PROGRAM UN01
VAR
	Ref_Unit: REFERENCE TO UDT_UnitAdmin;
	Ref_MachineStateModel: REFERENCE TO PackMlv3_StateModel;
	ref_Master1: REFERENCE TO UDT_AXISADMIN;	
	Cfg_ModeNames: ARRAY[0..31] OF STRING;
	Cfg_DisableStates: ARRAY [0..31] OF DINT;
	Cfg_ModeTransitions: ARRAY [0..31] OF DINT;
	HMI_O_StateCurrentName: STRING(255);
	HMI_O_ModeCurrentName: STRING(255);
	iHmiErr: INT;
	Loc_diEM_AbortingDone: DINT;
	Loc_diEM_ClearingDone: DINT;
	Loc_diEM_HoldingDone: DINT;
	Loc_diEM_ResettingDone: DINT;
	Loc_diEM_StartingDone: DINT;
	Loc_diEM_StoppingDone: DINT;
	Loc_diEM_SuspendingDone: DINT;
	Loc_diEM_UnSuspendingDone: DINT;
	Loc_diEM_UnHoldingDone: DINT;	
	Loc_diEM_Fault: DINT;
	Loc_diEM_Warning: DINT;	

	// 安全复位
	tonSafetyReset: TON;
	ft_SafetyReset: F_TRIG;
	iSafetyResetSeq: INT;	
	//EtherCat	
	iFaultClearSeq: INT;
	tonFaultClear: Ton;
	bClearAllFault: BOOL;
	xDebugReset: BOOL;
	arEventEmpty: ARRAY[1..256] OF BOOL;
	arSys1EventEmpty: ARRAY[1..20] OF BOOL;
	arSys2EventEmpty: ARRAY[21..40] OF BOOL;
	arSys3EventEmpty: ARRAY[1..20] OF BOOL;	
	loc_bAnyStopError: BOOL;
	j: INT;

	tonTimeHigh: TON;
	tonTimeLow: TON;
	arBlink: ARRAY[1..10] OF blink;
	
	tonFaultHandler: Ton;	
	StopEvent: ARRAY[0..40] OF UDT_EVENT;	
	arCylinder_AOI: ARRAY[1..80] OF AOI_CylinderAdmin;	
	arVacuum_AOI: ARRAY[1..60] OF AOI_VacuumAdmin;
    arSensor_AOI: ARRAY[1..60] OF AOI_Sensoradmin;	
	arHeat_AOI: ARRAY[1..8] OF Aoi_HeatBase;
    bUnitFS: BOOL;

	diUnitStopEvent0: DINT;
	rtWorkLocMode: R_trig;
	iRecipeSeq: INT;
	tonCmdReset: TON;
	tonCmdStart: TON;
	diSys1StopEvent1: DINT;
	diSys1StopEvent2: DINT;
	diSys2StopEvent1: DINT;
	diSys2StopEvent2: DINT;
	diSys3StopEvent1: DINT;
	diSys3StopEvent2: DINT;
	diSys3StopEvent3: DINT;
	rtAllaxisHomed: R_TRIG;
	tonRecipeSeq: Ton;
	
	tongeneralEvent0:ARRAY[0..255] OF Ton;

	diSys3StopEvent4: DINT;
	bSys1StopError: BOOL;
	bSys2StopError: BOOL;
	bSys3StopError: BOOL;

	iC: INT;
	
	arDropCylinder_AOI: ARRAY[1..40] OF AOI_CylinderAdmin;	
	iNotDone: INT;
	aoiActiveTotalTime: AOI_Timer;
	aoiWorkTotalTime: AOI_Timer;
	aoi10MinuteTime: AOI_Timer;
	
	rtGoodCount: R_TRIG;
	rtNoGoodCount: R_trig;
	rMaxCounterTime: DINT;
	rMaxDropTime: DINT;
	i: INT;
	iInitCnt: INT;
	iAutoCut: INT;
	tonAutoCut: Ton;
	iCutCnt: INT;
	bBoxRecipeUpdate: BOOL;
	bEn10Minute: BOOL;
	bReset10Minute: BOOL;
	diTransferCntOld: DINT;
	tonRecipeReset: Ton;
	bFirstCyclinderScan: BOOL;
	bAnySaftyDoorOpen: BOOL;
	tonCounterAirOpen: Ton;
END_VAR

VAR CONSTANT
   EM_OK: ARRAY[0..64] OF BOOL :=[65(0)];
   diEm_Done: DINT:=0;
END_VAR

//PLC IP地址IP 192.168.1.10 HMI1 IP 192.168.1.12 HMI2 IP 192.168.1.13 路由器 192.168.1.1 密码IPB19021 账号admin
//plc administrator 1 
//HMI 2222 
//激光打标机IP 192.168.1.20 
Ref_Unit REF=Unit01;
Ref_MachineStateModel REF= UN01_MachineStateModel;
ref_Master1 REF= arVirtualAxisAdmin[1];
CM02_ConditionsModules();
CM03_Cylinder();
CM04_Vacuum();
CM05_Sensor();
CM06_Heat();
CM07_Counters();
CM10_LightStatus();
SR02_Recipe();
UP01_PackML();
UP02_StateComplete();
EM01_Master();
EM02_Follower1();
EM03_Follower2();
EM04_FOllower3();
EM05_Counters();
EM06_Follower4_5();
EM07_Belt6();
EM08_Belt7();
SR91_OEE();
CM01_OperationLocal();
SR05_Manual();

IF NOT bUnitFS THEN
   SR01_Initialize();
END_IF

SR03_FaultHandler();
SR04_Parameter();
SR90_SafetyReset();
SR99_FaultClear();

DebugPro();

ACTION CM01_OperationLocal:
Ref_MachineStateModel.Cmd_Clear:=HMI_LocModeInput.ClearFault OR xDebugReset;
bAnySaftyDoorOpen:=arSafeDoorSts[19] OR arSafeDoorSts[20] OR arSafeDoorSts[21] OR arSafeDoorSts[22];
//前后设备急停串联
IF (glb_diEstopButton_UN01<>0) THEN
	Ref_MachineStateModel.Cmd_Abort:=TRUE;
	glb_AllAxisHomed_UN01:=FALSE;
	ELSE
	Ref_MachineStateModel.Cmd_Abort:=FALSE;
END_IF
//清除故障
IF Ref_MachineStateModel.Cmd_Clear THEN
   bClearAllFault:=TRUE;
END_IF
//停机
IF (HMI_LocModeInput.Stop OR glb_bStopButton_UN01) OR 
   (bAnySaftyDoorOpen AND Ref_MachineStateModel.Sts_Resetting) AND NOT Ref_MachineStateModel.Sts_Held THEN
	Ref_MachineStateModel.Cmd_Stop:=TRUE;
	ELSE
	Ref_MachineStateModel.Cmd_Stop:=FALSE;	
END_IF
//暂停
IF ((loc_bAnyStopError OR bAnySaftyDoorOpen) AND Ref_MachineStateModel.Sts_Execute) 
OR HMI_LocModeInput.Hold THEN
	Ref_MachineStateModel.Cmd_Hold:=TRUE;
	ELSE
	Ref_MachineStateModel.Cmd_Hold:=FALSE;	
END_IF
//启动
tonCmdStart(IN:= (HMI_LocModeInput.Start OR glb_bStartButton_UN01), PT:=T#2S , Q=> , ET=> );
IF tonCmdStart.Q AND glb_bAllSafetyOk 
AND NOT loc_bAnyStopError  
AND Ref_MachineStateModel.Sts_Idle
AND glb_bModeSwitch_UN01 THEN
	Ref_MachineStateModel.Cmd_Start:=TRUE;
	ELSE
	Ref_MachineStateModel.Cmd_Start:=FALSE;	
END_IF
//复位
tonCmdReset(IN:= (HMI_LocModeInput.Reset OR glb_bResetButton_UN01), PT:=T#2S , Q=> , ET=> );
IF tonCmdReset.Q AND NOT loc_bAnyStopError AND glb_bModeSwitch_UN01 THEN
   IF HMI_LocModeINPUT.Reset THEN
	  glb_AllAxisHomed_UN01:=FALSE;
   END_IF
   Ref_MachineStateModel.Cmd_Reset:=TRUE;
   ELSE
   Ref_MachineStateModel.Cmd_Reset:=FALSE;	 
END_IF

//安全复位
IF (glb_bResetButton_UN01 OR glb_bResetButton_UN02) AND
NOT glb_bAllSafetyOk THEN
   glb_bSafetyReset:=TRUE;
END_IF

//解除暂停
IF tonCmdStart.Q  AND Ref_MachineStateModel.Sts_Held  
AND glb_bModeSwitch_UN01 AND NOT loc_bAnyStopError THEN
	Ref_MachineStateModel.Cmd_UnHold:=TRUE;
	ELSE
    Ref_MachineStateModel.Cmd_UnHold:=FALSE;
END_IF

//等待启动
IF Ref_MachineStateModel.Sts_Idle THEN
	glb_AllAxisHomed_UN01:=TRUE;
END_IF
END_ACTION

ACTION CM02_ConditionsModules:
Loc_diEM_AbortingDone:=MEMCMP(pBuf1:=ADR(Ref_Unit.EM_Aborting_Done) , pBuf2:=ADR(Ref_Unit.EM_Selected) , n:=SIZEOF(Ref_Unit.EM_Selected));
Loc_diEM_ClearingDone:=MEMCMP(pBuf1:=ADR(Ref_Unit.EM_Clearing_Done) , pBuf2:=ADR(Ref_Unit.EM_Selected) , n:=SIZEOF(Ref_Unit.EM_Selected));
Loc_diEM_HoldingDone:=MEMCMP(pBuf1:=ADR(Ref_Unit.EM_Holding_Done) , pBuf2:=ADR(Ref_Unit.EM_Selected) , n:=SIZEOF(Ref_Unit.EM_Selected));
Loc_diEM_ResettingDone:=MEMCMP(pBuf1:=ADR(Ref_Unit.EM_Resetting_Done) , pBuf2:=ADR(Ref_Unit.EM_Selected) , n:=SIZEOF(Ref_Unit.EM_Selected));
Loc_diEM_StartingDone:=MEMCMP(pBuf1:=ADR(Ref_Unit.EM_Starting_Done) , pBuf2:=ADR(Ref_Unit.EM_Selected) , n:=SIZEOF(Ref_Unit.EM_Selected));
Loc_diEM_StoppingDone:=MEMCMP(pBuf1:=ADR(Ref_Unit.EM_Stopping_Done) , pBuf2:=ADR(Ref_Unit.EM_Selected) , n:=SIZEOF(Ref_Unit.EM_Selected));
Loc_diEM_SuspendingDone:=MEMCMP(pBuf1:=ADR(Ref_Unit.EM_Suspending_Done) , pBuf2:=ADR(Ref_Unit.EM_Selected) , n:=SIZEOF(Ref_Unit.EM_Selected));
Loc_diEM_UnSuspendingDone:=MEMCMP(pBuf1:=ADR(Ref_Unit.EM_UnSuspending_Done) , pBuf2:=ADR(Ref_Unit.EM_Selected) , n:=SIZEOF(Ref_Unit.EM_Selected));
Loc_diEM_UnHoldingDone:=MEMCMP(pBuf1:=ADR(Ref_Unit.EM_UnHolding_Done) , pBuf2:=ADR(Ref_Unit.EM_Selected) , n:=SIZEOF(Ref_Unit.EM_Selected));

Loc_diEM_Fault:=MEMCMP(pBuf1:=ADR(Ref_Unit.EM_Fault) , pBuf2:=ADR(EM_OK) , n:=SIZEOF(Ref_Unit.EM_Selected));
Loc_diEM_Warning:=MEMCMP(pBuf1:=ADR(Ref_Unit.EM_Warning) , pBuf2:=ADR(EM_OK) , n:=SIZEOF(Ref_Unit.EM_Selected));

Ref_Unit.EM_Selected:=HMI_EMSelectUn01;
END_ACTION

ACTION CM03_Cylinder:
FOR i:= 1 TO 60 DO
	arPackCylinder[i].i.CheckTime:=10000;
	arPackCylinder[i].i.Mode:=1;	
    arCylinder_AOI[i](Admin:= arPackCylinder[i]);
END_FOR
	arDropBufferCyclinder[1].i.CheckTime:=10000;
	arDropBufferCyclinder[1].i.Mode:=1;
	arDropBufferCyclinder[2].i.CheckTime:=10000;
	arDropBufferCyclinder[2].i.Mode:=1;
arCylinder_AOI[61](Admin:= arDropBufferCyclinder[1]);
arCylinder_AOI[62](Admin:= arDropBufferCyclinder[2]);
IF NOT bFirstCyclinderScan THEN
   bFirstCyclinderScan:=TRUE;
END_IF
END_ACTION

ACTION CM04_Vacuum:
FOR i:=1 TO 60 DO
	arPackVacuum[i].i.CheckTime:=5000;
	arPackVacuum[i].i.BlowTime:=1000;
	arVacuum_AOI[i](admin:= arPackVacuum[i]);
END_FOR
END_ACTION

ACTION CM05_Sensor:
FOR i:=1 TO 60 DO
	arSensor_AOI[i](Admin:=arPackSensor[i] );
END_for
END_ACTION

ACTION CM06_Heat:
	arHeat_AOI[1](	Enable:=NOT HMI_HeatDisable , 	PV:=HMI_HeatTempAct[1] , 	SV:= HMI_HeatTempSet[1], 
 	Reset:= ,HighLimit:= 30,lowLimit:= 30,MaxLimit:=300,Kp:=20,Ki:=0.5,Kd:=3,
	Active=> arPackHeatRealy[1], 
	Error=> );
	arHeat_AOI[2](	Enable:=NOT HMI_HeatDisable , 	PV:=HMI_HeatTempAct[2] , 	SV:= HMI_HeatTempSet[2], 
	Reset:= ,HighLimit:= 30, lowLimit:= 30,MaxLimit:=300,Kp:=20,Ki:=0.5,Kd:=3,
	Active=> arPackHeatRealy[2], 
	Error=> );
	arHeat_AOI[3](	Enable:=NOT HMI_HeatDisable , 	PV:=HMI_HeatTempAct[3] , 	SV:= HMI_HeatTempSet[3], 
    Reset:= ,HighLimit:= 30, lowLimit:= 30,MaxLimit:=300,Kp:=20,Ki:=0.5,Kd:=3,
	Active=> arPackHeatRealy[3], 
	Error=> );
	arHeat_AOI[4](	Enable:=NOT HMI_HeatDisable , 	PV:=HMI_HeatTempAct[4] , 	SV:= HMI_HeatTempSet[4], 
    Reset:= ,HighLimit:= 30, lowLimit:= 30,MaxLimit:=300,Kp:=20,Ki:=0.5,Kd:=3,		
	Active=> arPackHeatRealy[4], 
	Error=> );
	arHeat_AOI[5](	Enable:=NOT HMI_HeatDisable , 	PV:=HMI_HeatTempAct[5] , 	SV:= HMI_HeatTempSet[5], 
    Reset:= ,HighLimit:= 30, lowLimit:= 30,MaxLimit:=300,Kp:=20,Ki:=0.5,Kd:=3,		
	Active=> arPackHeatRealy[5], 
	Error=> );
	arHeat_AOI[6](	Enable:=NOT HMI_HeatDisable , 	PV:=HMI_HeatTempAct[6] , 	SV:= HMI_HeatTempSet[6],
    Reset:= ,HighLimit:= 30, lowLimit:= 30,MaxLimit:=300,Kp:=20,Ki:=0.5,Kd:=3, 
	Active=> arPackHeatRealy[6], 
	Error=> );
	arHeat_AOI[7](	Enable:=NOT HMI_HeatDisable , 	PV:=HMI_HeatTempAct[7] , 	SV:= HMI_HeatTempSet[7],
    Reset:= ,HighLimit:= 30, lowLimit:= 30,MaxLimit:=300,Kp:=20,Ki:=0.5,Kd:=3, 
	Active=> arPackHeatRealy[7], 
	Error=> );
	arHeat_AOI[8](	Enable:=NOT HMI_HeatDisable , 	PV:=HMI_HeatTempAct[8] , 	SV:= HMI_HeatTempSet[8],
    Reset:= ,HighLimit:= 30, lowLimit:= 30,MaxLimit:=300,Kp:=20,Ki:=0.5,Kd:=3, 
	Active=> arPackHeatRealy[8], 
	Error=> );	
	
	HMI_HeatTempAct[1]:=INT_TO_REAL(EL3312[1,1].Value)/10;
	HMI_HeatTempAct[2]:=INT_TO_REAL(EL3312[1,2].Value)/10;
	HMI_HeatTempAct[3]:=INT_TO_REAL(EL3312[2,1].Value)/10;
	HMI_HeatTempAct[4]:=INT_TO_REAL(EL3312[2,2].Value)/10;
	HMI_HeatTempAct[5]:=INT_TO_REAL(EL3312[3,1].Value)/10;
	HMI_HeatTempAct[6]:=INT_TO_REAL(EL3312[3,2].Value)/10;   
	HMI_HeatTempAct[7]:=INT_TO_REAL(EL3312[4,1].Value)/10;
	HMI_HeatTempAct[8]:=INT_TO_REAL(EL3312[4,2].Value)/10;
END_ACTION

ACTION CM07_Counters:
iInitCnt:=0;
rMaxDropTime:=0;
rMaxCounterTime:=0;
FOR ic:=1 TO 10 DO
	arCounters[iC](
		In_Total:= RecipeBuffer.amount, 
		Quantity:= RecipeBuffer.Counters[iC].Quantity, 
		ProcessTime=> HMI_OEEView.CounterProcessTime[iC] ,
		Axis:= arRealAxisAdmin[iC], 
		Checktime:= HMI_CntCheckTime,
		DropSensor:= arDropSensor[iC], 
		LowSensor:= arLowSensor[iC], 
		HighSensor:= arhighSensor[iC],
		DropFlag:= glb_BinBelt1.bin[iC].arDrop[iC],
		Cylinder:= arDropCylinder[iC]);	
END_FOR
FOR ic:=11 TO 20 DO
	arCounters[iC](
		In_Total:= RecipeBuffer.amount, 
		Quantity:= RecipeBuffer.Counters[iC].Quantity,
       	CheckTime:= 1500,
		ProcessTime=> HMI_OEEView.CounterProcessTime[iC] ,
		Axis:= arRealAxisAdmin[iC], 
		Checktime:= HMI_CntCheckTime,
		DropSensor:= arDropSensor[iC], 
		LowSensor:= arLowSensor[iC], 
		HighSensor:= arhighSensor[iC],
		DropFlag:= glb_BinBelt1.bin[iC+20].arDrop[iC+20],
		Cylinder:= arDropCylinder[iC]);	
END_FOR

FOR ic:=21 TO 30 DO
	arCounters[iC](
		In_Total:= RecipeBuffer.amount, 
		Quantity:= RecipeBuffer.Counters[iC].Quantity, 
		ProcessTime=> HMI_OEEView.CounterProcessTime[iC] ,
		Axis:= arRealAxisAdmin[iC], 
		Checktime:= HMI_CntCheckTime,
		DropSensor:= arDropSensor[iC], 
		LowSensor:= arLowSensor[iC], 
		HighSensor:= arhighSensor[iC],
		DropFlag:= glb_BinBelt2.bin[ic-20].arDrop[iC-20],
		Cylinder:= arDropCylinder[iC]);	
END_FOR

FOR ic:=31 TO 40 DO
	arCounters[iC](
		In_Total:= RecipeBuffer.amount, 
		Quantity:= RecipeBuffer.Counters[iC].Quantity, 
		ProcessTime=> HMI_OEEView.CounterProcessTime[iC] ,
		Axis:= arRealAxisAdmin[iC], 
		Checktime:= HMI_CntCheckTime,
		DropSensor:= arDropSensor[iC], 
		LowSensor:= arLowSensor[iC], 
		HighSensor:= arhighSensor[iC],
		DropFlag:= glb_BinBelt2.bin[iC].arDrop[iC],
		Cylinder:= arDropCylinder[iC]);	
END_FOR
  
FOR iC:=1 TO 40 DO
	arDropCylinder_AOI[iC](Admin:= arDropCylinder[iC]);
	arDropCylinder[iC].i.CheckTime:=1500;
	arDropCylinder[iC].i.Mode:=1;	
   IF NOT  arCounters[iC].Busy THEN
      IF rMaxCounterTime < arCounters[iC].ProcessTime THEN
		 rMaxCounterTime:= arCounters[iC].ProcessTime;
	  END_IF
   END_IF  
   arCounters[iC].SkipAlarm:=HMI_SkipCntAlarm[iC];
   arCounters[iC].CheckCnt:=HMI_CntCheck[iC];
   HMI_CountersCntUp[ic]:=arCounters[iC].CntUp;
   
   HMI_OEEView.DropProcessTime[ic]:=(arDropCylinder_AOI[iC].ActInTime+arDropCylinder_AOI[iC].ActOutTime)/2;
   IF rMaxDropTime<HMI_OEEView.DropProcessTime[ic] THEN
	  rMaxDropTime:=HMI_OEEView.DropProcessTime[ic];  
   END_IF
END_FOR
END_ACTION

ACTION CM10_LightStatus:

IF glb_bAllSafetyOk THEN
	glb_bResetBottonLight_UN01:=TRUE;
	ELSE 
    glb_bResetBottonLight_UN01:=arBlink[1].OUT;
END_IF

{region Lihgtsys1} 
//红灯
glb_arLightRed_UN01[1]:=Ref_MachineStateModel.Sts_Aborted OR Ref_MachineStateModel.Sts_Aborting OR (arblink[1].OUT AND bSys1StopError);
glb_arLightAlarm_UN01[1]:=(glb_arLightRed_UN01[1] OR glb_arLightYellow_UN01[1]) AND NOT HMI_AlarmMute;
//绿灯	  
glb_arLightGreen_UN01[1]:= Ref_MachineStateModel.Sts_Execute OR  Ref_MachineStateModel.Sts_Stopping OR
( arblink[1].OUT AND NOT bSys1StopError  AND NOT Ref_MachineStateModel.Sts_Aborted AND NOT Ref_MachineStateModel.Sts_Resetting
AND( Ref_MachineStateModel.Sts_Stopped OR Ref_MachineStateModel.Sts_Idle OR Ref_MachineStateModel.Sts_Held))
OR (Ref_MachineStateModel.Sts_Resetting  AND arblink[2].OUT);	 
//黄灯
glb_arLightYellow_UN01[1]:= (HMI_GeneralEvent[2].ID[1] OR HMI_GeneralEvent[2].ID[2] OR HMI_GeneralEvent[2].ID[3] OR HMI_GeneralEvent[2].ID[4]
OR HMI_GeneralEvent[2].ID[5] OR HMI_GeneralEvent[2].ID[6] OR HMI_GeneralEvent[2].ID[7] OR HMI_GeneralEvent[2].ID[8] OR HMI_GeneralEvent[2].ID[9]
OR HMI_GeneralEvent[2].ID[10] OR HMI_GeneralEvent[2].ID[11] OR HMI_GeneralEvent[2].ID[12] OR HMI_GeneralEvent[2].ID[13] OR HMI_GeneralEvent[2].ID[14]
OR HMI_GeneralEvent[2].ID[15] OR HMI_GeneralEvent[2].ID[16] OR HMI_GeneralEvent[2].ID[17] OR HMI_GeneralEvent[2].ID[18] OR HMI_GeneralEvent[2].ID[19]
OR HMI_GeneralEvent[2].ID[20]) AND arblink[1].OUT;	 	 
		  
(*照明灯*)  
glb_arLightRelay_UN01[1]:= arSafeDoorSts[1] OR arSafeDoorSts[2] OR arSafeDoorSts[3] OR arSafeDoorSts[4] OR
arSafeDoorSts[5] OR arSafeDoorSts[6] OR arSafeDoorSts[7] OR arSafeDoorSts[8] OR
arSafeDoorSts[9] ;
	   
{end_region}				
{region Lihgtsys2} 					 

glb_arLightRed_UN01[2]:=Ref_MachineStateModel.Sts_Aborted OR Ref_MachineStateModel.Sts_Aborted OR ( arblink[1].OUT AND bSys2StopError );
glb_arLightAlarm_UN01[2]:=(glb_arLightRed_UN01[2] OR glb_arLightYellow_UN01[2]) AND NOT HMI_AlarmMute;
		  
glb_arLightGreen_UN01[2]:= Ref_MachineStateModel.Sts_Execute OR Ref_MachineStateModel.Sts_Stopping OR
( arblink[1].OUT AND NOT bSys2StopError  AND NOT Ref_MachineStateModel.Sts_Aborted AND NOT Ref_MachineStateModel.Sts_Resetting
AND( Ref_MachineStateModel.Sts_Stopped OR Ref_MachineStateModel.Sts_Idle OR Ref_MachineStateModel.Sts_Held))
OR (Ref_MachineStateModel.Sts_Resetting  AND arblink[2].OUT);
 
//黄灯
glb_arLightYellow_UN01[2]:= (HMI_GeneralEvent[2].ID[21] OR HMI_GeneralEvent[2].ID[22] OR HMI_GeneralEvent[2].ID[23] OR HMI_GeneralEvent[2].ID[24]
OR HMI_GeneralEvent[2].ID[25] OR HMI_GeneralEvent[2].ID[26] OR HMI_GeneralEvent[2].ID[27] OR HMI_GeneralEvent[2].ID[28] OR HMI_GeneralEvent[2].ID[29]
OR HMI_GeneralEvent[2].ID[30] OR HMI_GeneralEvent[2].ID[31] OR HMI_GeneralEvent[2].ID[32] OR HMI_GeneralEvent[2].ID[33] OR HMI_GeneralEvent[2].ID[34]
OR HMI_GeneralEvent[2].ID[35] OR HMI_GeneralEvent[2].ID[36] OR HMI_GeneralEvent[2].ID[37] OR HMI_GeneralEvent[2].ID[38] OR HMI_GeneralEvent[2].ID[39]
OR HMI_GeneralEvent[2].ID[40]) AND arblink[1].OUT;		   
(*照明灯*)

glb_arLightRelay_UN01[2]:=arSafeDoorSts[10] OR arSafeDoorSts[11] OR arSafeDoorSts[12] OR arSafeDoorSts[13] OR
arSafeDoorSts[14] OR arSafeDoorSts[15] OR arSafeDoorSts[16] OR arSafeDoorSts[17] OR
arSafeDoorSts[18] ;
	  
{end_region}		   

{region Lihgtsys3} 	

glb_arLightRed_UN01[3]:=Ref_MachineStateModel.Sts_Aborted OR Ref_MachineStateModel.Sts_Aborted OR (arblink[1].OUT AND bSys3StopError);
glb_arLightAlarm_UN01[3]:=glb_arLightRed_UN01[3] AND NOT HMI_AlarmMute;
			   
							  
glb_arLightGreen_UN01[3]:= Ref_MachineStateModel.Sts_Execute OR Ref_MachineStateModel.Sts_Stopping OR
( arblink[1].OUT AND NOT bSys3StopError  AND NOT Ref_MachineStateModel.Sts_Aborted AND NOT Ref_MachineStateModel.Sts_Resetting
AND( Ref_MachineStateModel.Sts_Stopped OR Ref_MachineStateModel.Sts_Idle OR Ref_MachineStateModel.Sts_Held))
OR (Ref_MachineStateModel.Sts_Resetting  AND arblink[2].OUT);
//黄灯
glb_arLightYellow_UN01[3]:= ( HMI_GeneralEvent[0].ID[1] OR HMI_GeneralEvent[0].ID[2] ) AND arblink[1].OUT;		   
(*照明灯*)

{end_region}

arBlink[1](TimeH:=100 , TimeL:=1000 , OUT=> );
arBlink[2](TimeH:=200 , TimeL:=200 , OUT=> );
END_ACTION

ACTION SR01_Initialize:
glb_bCounterAirValve_UN01:=TRUE;
bUnitFS:=TRUE;
HMI_EMSelectUN01[1]:=TRUE;
HMI_EMSelectUN01[2]:=TRUE;
HMI_EMSelectUN01[3]:=TRUE;
HMI_EMSelectUN01[4]:=TRUE;
HMI_EMSelectUN01[5]:=TRUE;
HMI_EMSelectUN01[6]:=TRUE;
HMI_EMSelectUN01[7]:=TRUE;
HMI_EMSelectUN01[8]:=TRUE;
	
;
END_ACTION

ACTION SR02_Recipe:
rtWorkLocMode(CLK:=HMI_LocModeEnable , Q=> );
rtAllaxisHomed(CLK:= glb_AllAxisHomed_UN01, Q=> );
tonRecipeReset(IN:=glb_bResetButton_UN01 AND Ref_MachineStateModel.Sts_Execute , PT:= T#5S , Q=> , ET=> );

CASE iRecipeSeq OF 
	0: 
	   HMI_RecipeReset:=TRUE;
	   bBoxRecipeUpdate:=FALSE;
       IF  glb_AllAxisHomed_UN01  THEN
		   IF HMI_LocModeEnable THEN
			  iRecipeSeq:=10;
		   END_IF
		   IF Hmi_Input.ModifyRecipe OR tonRecipeReset.Q THEN 
			  iRecipeSeq:=20;
			  HMI_RecipeReset:=FALSE;
		   END_IF
		   IF HMI_RecipeRedo THEN
			  HMI_RecipeReset:=FALSE;
			  iRecipeSeq:=300;  
		   END_IF
		   IF HMI_RecipCancel THEN
			  HMI_RecipeReset:=FALSE;
			  iRecipeSeq:=200;  
		   END_IF
	   END_IF
	
	10:(*本地模拟生产配方*)
        Hmi_Output.InQuantity:=49;
		Hmi_Output.OutQuantity:=0;
		FOR i:=1 TO 40 DO
			Hmi_Output.Counters[i].Quantity:=5;
			Hmi_Output.Counters[i].ID:=i;
		END_FOR
	    iRecipeSeq:=90;	


     20:
        (**生产任务配方**)
		IF Hmi_Recipe.amount<>0 THEN//配方有效
			RecipeBuffer:=HMI_RECIPE;
			RecipeBuffer.user:=HMI_RECIPE.user;
			Hmi_Output.InQuantity:=RecipeBuffer.amount;
			Hmi_Output.OutQuantity:=0;
			FOR i:=1 TO 40 DO
				Hmi_Output.Counters[i].Quantity:=RecipeBuffer.Counters[i].Quantity;
				Hmi_Output.Counters[i].ID:=RecipeBuffer.Counters[i].ID;
			END_FOR
			iRecipeSeq:=90;	
		ELSE//配方无效
            iRecipeSeq:=200;	
		END_IF
 

		
	90: //复位料仓
        Glb_BinList.Reset:=TRUE;
		FOR i:=1 TO 40 DO
		    arCounters[i].Reset:=TRUE;
		END_FOR 
	    iRecipeSeq:=91;
    91: //复位数粒 		
		FOR i:=1 TO 40 DO
		    arCounters[i].Reset:=FALSE;
		END_FOR
		Glb_BinList.Reset:=FALSE;
		glb_lrMasterTargetCnt:=glb_lrMasterTargetCnt + Hmi_Output.InQuantity;
		glb_lrBelt1TargetCnt:=glb_lrBelt1TargetCnt + Hmi_Output.InQuantity + HMI_B1DropBinNo;
		glb_lrBelt2Targetcnt:=glb_lrBelt2Targetcnt + Hmi_Output.InQuantity + HMI_B2DropBinNo;
		glb_lrBelt3Targetcnt:=glb_lrBelt3Targetcnt+ Hmi_Output.InQuantity + HMI_B3DropBinNo3;	
		iRecipeSeq:=92;
		
	92:	
	    tonRecipeSeq(IN:=TRUE, PT:=T#1S , Q=> , ET=> );
		IF tonRecipeSeq.Q THEN
	       tonRecipeSeq(IN:=FALSE, PT:=T#1S , Q=> , ET=> );	
			HMI_Output.RecipeComplete:=FALSE;
			Hmi_Input.ModifyRecipe:=FALSE;
			HMI_Output.RecipeModifyDone:=TRUE;	  	  
            iRecipeSeq:=93;	
		END_IF	
		
	93:
        tonRecipeSeq(IN:=TRUE, PT:=T#1S , Q=> , ET=> );
		IF tonRecipeSeq.Q THEN
	       tonRecipeSeq(IN:=FALSE, PT:=T#1S , Q=> , ET=> );	  	  
           iRecipeSeq:=100;	
		END_IF	
	 
	100:
	    glb_BinBelt1.bin[1].Name:=RecipeBuffer.user;
		glb_BinBelt1.bin[1].Amount:=RecipeBuffer.amount;//获取生产数量
	    HMI_RecipeAbort:=FALSE;
        Hmi_Output.RecipeEmplty:=FALSE;
		IF glb_lrBelt1wrkCnt>14  AND NOT bBoxRecipeUpdate  THEN
		   glb_lrBoxTargetCnt := glb_lrBoxTargetCnt+Hmi_Output.InQuantity/7;
		   bBoxRecipeUpdate:=TRUE;
		END_IF

		IF glb_lrBelt1wrkCnt = glb_lrBelt1TargetCnt AND glb_lrBelt2wrkCnt = glb_lrBelt2TargetCnt THEN
			HMI_Output.RecipeComplete:=TRUE;
		END_IF
		
	    IF HMI_Output.RecipeComplete THEN
		   HMI_Output.RecipeModifyDone:=FALSE;
	       iRecipeSeq:=110;
		   ELSE IF NOT glb_AllAxisHomed_UN01 THEN//配方被中止
			           HMI_RecipeAbort:=TRUE;
					   iRecipeSeq:=900;
		        END_IF
		END_IF
		
    
    110:
	    tonRecipeSeq(IN:=TRUE, PT:=T#1S , Q=> , ET=> );
		IF tonRecipeSeq.Q THEN
	       tonRecipeSeq(IN:=FALSE, PT:=T#1S , Q=> , ET=> );	
           iRecipeSeq:=0;		
		END_IF
		
(***************************************************************)		
    200: 
        HMI_RecipeAbort:=FALSE;
	    tonRecipeSeq(IN:=TRUE, PT:=T#1S , Q=> , ET=> );
		IF tonRecipeSeq.Q THEN
	       tonRecipeSeq(IN:=FALSE, PT:=T#1S , Q=> , ET=> );	
			HMI_Output.RecipeComplete:=FALSE;
			Hmi_Input.ModifyRecipe:=FALSE;
			HMI_Output.RecipeModifyDone:=TRUE;	  	  
           iRecipeSeq:=210;	
		END_IF	
    210:
	    tonRecipeSeq(IN:=TRUE, PT:=T#1S , Q=> , ET=> );
		IF tonRecipeSeq.Q THEN
	       tonRecipeSeq(IN:=FALSE, PT:=T#1S , Q=> , ET=> );	
			HMI_Output.RecipeComplete:=TRUE;
			HMI_Output.RecipeModifyDone:=FALSE;	  	  
           iRecipeSeq:=220;	
		END_IF	

    220:
	    tonRecipeSeq(IN:=TRUE, PT:=T#1S , Q=> , ET=> );
		IF tonRecipeSeq.Q THEN
	       tonRecipeSeq(IN:=FALSE, PT:=T#1S , Q=> , ET=> );		  	  
           iRecipeSeq:=0;	
		END_IF	
(***********************************************************)		
	300:
		IF RecipeBuffer.amount<>0 THEN
			Hmi_Output.InQuantity:=RecipeBuffer.amount;
			Hmi_Output.OutQuantity:=0;
			FOR i:=1 TO 40 DO
				Hmi_Output.Counters[i].Quantity:=RecipeBuffer.Counters[i].Quantity;
				Hmi_Output.Counters[i].ID:=RecipeBuffer.Counters[i].ID;
			END_FOR
			iRecipeSeq:=90;	
		ELSE
            iRecipeSeq:=200;	
		END_IF	
			
	900:
	    Hmi_Output.InQuantity:=0;
		Hmi_Output.OutQuantity:=0;
		Hmi_Output.RecipeEmplty:=TRUE;
		HMI_Output.RecipeModifyDone:=FALSE;
		HMI_Output.RecipeComplete:=FALSE;

        FOR i:=1 TO 40 DO
		    arCounters[i].Reset:=TRUE;	
		END_FOR
	    Glb_BinList.Reset:=TRUE;
	 	iRecipeSeq:=1000;
	1000:
        HMI_Output.RecipeComplete:=FALSE;
		HMI_Output.RecipeModifyDone:=FALSE;	
		Glb_BinList.Reset:=FALSE;
		FOR i:=1 TO 40 DO
		    arCounters[i].Reset:=FALSE;	
		END_FOR
		
		iRecipeSeq:=0;
END_CASE
END_ACTION

ACTION SR03_FaultHandler:
tonFaultHandler(IN:=glb_bDevice1AllOP AND  glb_bAllSafetyOk, PT:= T#2S, Q=> , ET=> );
//停机故障信息(0,1 安全类报警)(2,3通讯类报警), (4,5,6,7伺服类报警)(8,9,10,11变频器类报警)
//(12,13,14,15气缸类报警)(16,17,18,19传感器类报警)(20,21,22,23真空类报警)(24...其它类报警) 
HMI_StopEvent[0].ID[1]:= NOT glb_bDevice1AllOP;//数粒Ethercat报警
HMI_StopEvent[0].ID[2]:= FALSE;//装罐Ethercat报警
HMI_StopEvent[0].ID[3]:= NOT glb_arSafeRelayNo_UN01[1];//安全继电器吸合报警		
HMI_StopEvent[0].ID[5]:= FALSE;	//机器人报警
HMI_StopEvent[0].ID[6]:= FALSE;//喷码机报警
HMI_StopEvent[0].ID[7]:= glb_MembraneAlarm;//

FOR iHmiErr:=1 TO 8 DO
	HMI_StopEvent[5].ID[iHmiErr]:=arHeat_AOI[iHmiErr].Error; //加热1—-8温度报警
END_FOR  

IF tonFaultHandler .Q THEN	
    HMI_StopEvent[0].ID[4]:= FALSE;			
    HMI_StopEvent[0].ID[8]:= NOT glb_bAirFeedback_UN01[1];//数粒系统气压异常报警
    HMI_StopEvent[0].ID[9]:= NOT glb_bAirFeedback_UN01[2];//装罐系统气压异常报警
    HMI_StopEvent[0].ID[10]:= arDropBufferCyclinder[1].o.Error;
	HMI_StopEvent[0].ID[11]:= arDropBufferCyclinder[2].o.Error;
	
	FOR iHmiErr:=1 TO 64 DO//伺服报警
	   HMI_StopEvent[1].ID[iHmiErr]:=arRealAxisAdmin[iHmiErr].o.Error OR (arErrorCodeDrive[iHmiErr]<>0);
	END_FOR
	
	FOR iHmiErr:=1 TO 40 DO//落料气缸报警
		HMI_StopEvent[2].ID[iHmiErr]:=arDropCylinder[iHmiErr].o.Error;
	END_FOR
	
	FOR iHmiErr:=1 TO 50 DO//气缸报警
		HMI_StopEvent[3].ID[iHmiErr]:=arPackCylinder[iHmiErr].o.Error;
	END_FOR
	
	FOR iHmiErr:=1 TO 40 DO//真空报警
		HMI_StopEvent[4].ID[iHmiErr]:=arPackVacuum[iHmiErr].o.Error;
	END_FOR
	
	FOR iHmiErr:=1 TO 40 DO//数粒报警
		HMI_StopEvent[6].ID[iHmiErr]:=arCounters[iHmiErr].Error;
	END_FOR
			
	FOR iHmiErr:=1 TO 40 DO//安全门报警
		HMI_GeneralEvent[1].ID[iHmiErr]:= arSafeDoorSts[iHmiErr];
	END_FOR    
	FOR iHmiErr:=1 TO 40 DO
	    HMI_GeneralEvent[2].ID[iHmiErr]:= arCounters[iHmiErr].Warning ;// 暂时屏蔽
    END_FOR  
END_IF

tongeneralEvent0[1](IN:=NOT arPackSensor[1].o.Value OR NOT arPackSensor[2].o.Value 
OR NOT arPackSensor[3].o.Value OR NOT arPackSensor[4].o.Value 
OR NOT arPackSensor[5].o.Value OR NOT arPackSensor[6].o.Value OR NOT arPackSensor[7].o.Value , 
PT:=T#3S , Q=> , ET=> );

HMI_GeneralEvent[0].ID[1]:=tongeneralEvent0[1].Q; //铝杯工位1缺料

tongeneralEvent0[2](IN:=NOT arPackSensor[8].o.Value OR NOT arPackSensor[9].o.Value 
OR NOT arPackSensor[10].o.Value OR NOT arPackSensor[11].o.Value 
OR NOT arPackSensor[12].o.Value OR NOT arPackSensor[13].o.Value OR NOT arPackSensor[14].o.Value , 
PT:=T#3S , Q=> , ET=> );

HMI_GeneralEvent[0].ID[2]:=tongeneralEvent0[2].Q ; //铝杯工位2缺料

tongeneralEvent0[3](IN:=NOT arPackSensor[22].o.Value	 , 
PT:=T#10S , Q=> , ET=> );  
HMI_GeneralEvent[0].ID[3]:=NOT HMI_PrinterConnected; //打印机未启用
HMI_GeneralEvent[0].ID[4]:=HMI_PrinterFault; //打印机未启用
tongeneralEvent0[4](IN:= arPackCylinder[22].i.InSensor AND NOT arPackSensor[20].o.Value 
AND (arPackMotor[3].Backward OR	arPackMotor[3].Forward) , 
PT:=T#10S , Q=> , ET=> );  



//////////////////////////////////////////////////////////////////////////////////
//////////////**********************************************************//////////
//////////////**********************************************************//////////
//////////////**********************************************************//////////
//////////////**********************************************************//////////
//////////////////////////////////////////////////////////////////////////////////
IF tonFaultHandler .Q THEN	
   		 
	FOR i:=1 TO 20 DO
		StopEvent[1].ID[i]:=arRealAxisAdmin[i].o.Error;//数粒伺服1-20报警
	END_FOR	
	FOR i:=1 TO 20 DO
		StopEvent[2].ID[i]:=arDropCylinder[i].o.Error;//数粒气缸21-40报警
	END_FOR

	FOR i:=21 TO 40 DO
		StopEvent[3].ID[i]:=arRealAxisAdmin[i].o.Error;//数粒伺服1-20报警
	END_FOR	
		 StopEvent[3].ID[40]:=FALSE;
	FOR i:=21 TO 40 DO
		StopEvent[4].ID[i]:=arDropCylinder[i].o.Error;//数粒气缸21-40报警
	END_FOR
         
	FOR i:=41 TO 48 DO //后段设备被取消 48台伺服 20210420
		StopEvent[5].ID[i]:=arRealAxisAdmin[i].o.Error; //伺服41-47报警  48报警
	END_FOR	
	FOR i:=1 TO 20 DO
		StopEvent[6].ID[i]:=arPackCylinder[i].o.Error;
	END_FOR
        StopEvent[6].ID[41]:=arPackCylinder[41].o.Error;
		
	FOR i:=1 TO 20 DO
		StopEvent[7].ID[i]:=arPackVacuum[i].o.Error;
	END_FOR		
		 
	FOR i:=1 TO 8 DO
		StopEvent[8].ID[i]:=arHeat_AOI[i].Error;
	END_FOR					  
		 
END_IF
StopEvent[8].ID[20]:=HMI_StopEvent[5].ID[20];	 
StopEvent[8].ID[21]:=HMI_StopEvent[5].ID[21];	
StopEvent[8].ID[22]:=HMI_StopEvent[5].ID[22];	
StopEvent[8].ID[23]:=HMI_StopEvent[5].ID[23];	
StopEvent[8].ID[24]:=HMI_StopEvent[5].ID[24];	
StopEvent[8].ID[25]:=HMI_StopEvent[5].ID[25];	
StopEvent[8].ID[26]:=HMI_StopEvent[5].ID[26];	
		  
StopEvent[0].ID[1]:= NOT glb_bDevice1AllOP;
StopEvent[0].ID[2]:= glb_MembraneAlarm;
StopEvent[0].ID[3]:= NOT glb_arSafeRelayNo_UN01[1];	
StopEvent[0].ID[4]:= NOT glb_bAirFeedback_UN01[1];	
StopEvent[0].ID[5]:= NOT glb_bAirFeedback_UN01[2];	
StopEvent[0].ID[6]:= HMI_PrinterFault;
StopEvent[0].ID[7]:= arDropBufferCyclinder[1].o.Error;
StopEvent[0].ID[8]:= arDropBufferCyclinder[2].o.Error;
	 
diUnitStopEvent0:=MEMCMP(pBuf1:=ADR(StopEvent[0]) , pBuf2:=ADR(arEventEmpty) , n:=SIZEOF(arEventEmpty));
diSys1StopEvent1:=MEMCMP(pBuf1:=ADR(StopEvent[1]) , pBuf2:=ADR(arEventEmpty) , n:=SIZEOF(arEventEmpty));
diSys1StopEvent2:=MEMCMP(pBuf1:=ADR(StopEvent[2]) , pBuf2:=ADR(arEventEmpty) , n:=SIZEOF(arEventEmpty));	 
diSys2StopEvent1:=MEMCMP(pBuf1:=ADR(StopEvent[3]) , pBuf2:=ADR(arEventEmpty) , n:=SIZEOF(arEventEmpty));
diSys2StopEvent2:=MEMCMP(pBuf1:=ADR(StopEvent[4]) , pBuf2:=ADR(arEventEmpty) , n:=SIZEOF(arEventEmpty));		  
diSys3StopEvent1:=MEMCMP(pBuf1:=ADR(StopEvent[5]) , pBuf2:=ADR(arEventEmpty) , n:=SIZEOF(arEventEmpty));
diSys3StopEvent2:=MEMCMP(pBuf1:=ADR(StopEvent[6]) , pBuf2:=ADR(arEventEmpty) , n:=SIZEOF(arEventEmpty));			   
diSys3StopEvent3:=MEMCMP(pBuf1:=ADR(StopEvent[7]) , pBuf2:=ADR(arEventEmpty) , n:=SIZEOF(arEventEmpty));	
diSys3StopEvent4:=MEMCMP(pBuf1:=ADR(StopEvent[8]) , pBuf2:=ADR(arEventEmpty) , n:=SIZEOF(arEventEmpty));

IF diSys1StopEvent1=0 AND diSys1StopEvent2=0 THEN
   bSys1StopError:=FALSE;
ELSE
   bSys1StopError:=TRUE;	
END_IF
	
IF diSys2StopEvent1=0 AND diSys2StopEvent2=0 THEN
   bSys2StopError:=FALSE;
ELSE
   bSys2StopError:=TRUE;	
END_IF 
		  
IF 	 diSys3StopEvent1=0 AND diSys3StopEvent2=0 AND diSys3StopEvent3=0 AND diSys3StopEvent3=0 AND diSys3StopEvent4=0
AND diUnitStopEvent0=0 THEN		
    bSys3StopError:=FALSE;
ELSE
    bSys3StopError:=TRUE;	
END_IF
					
IF bSys1StopError OR bSys2StopError OR bSys3StopError THEN
   loc_bAnyStopError:=TRUE;
   ELSE
   loc_bAnyStopError:=FALSE; 
END_IF
END_ACTION

ACTION SR04_Parameter:
arVirtualAxisAdmin[1].i.Vel:=HMI_MasterVelo;

//数粒伺服
FOR i:=1 TO 40 DO 
	arRealAxisAdmin[i].i.Vel:=HMI_CountersVelo;
	arRealAxisAdmin[i].i.Acc:=HMI_CountersAcc;
	arRealAxisAdmin[i].i.Dec:=HMI_CountersDec;
	arRealAxisAdmin[i].i.Jerk:=HMI_CountersDec*100;
END_FOR
//皮带1
arRealAxisAdmin[41].i.Vel:=HMI_BeltVelo[1];
arRealAxisAdmin[41].i.Acc:=HMI_BeltAcc[1];
arRealAxisAdmin[41].i.Dec:=HMI_BeltDec[1];
arRealAxisAdmin[41].i.HomeOffset:=HMI_HomeOffsetBelt[1];
//皮带2
arRealAxisAdmin[42].i.Vel:=HMI_BeltVelo[2];
arRealAxisAdmin[42].i.Acc:=HMI_BeltAcc[2];
arRealAxisAdmin[42].i.Dec:=HMI_BeltDec[2];
arRealAxisAdmin[42].i.HomeOffset:=HMI_HomeOffsetBelt[2];
//皮带3
arRealAxisAdmin[43].i.Vel:=HMI_BeltVelo[3];
arRealAxisAdmin[43].i.Acc:=HMI_BeltAcc[3];
arRealAxisAdmin[43].i.Dec:=HMI_BeltDec[3];
arRealAxisAdmin[43].i.HomeOffset:=HMI_HomeOffsetBelt[3];
//皮带4 //皮带5

//皮带6
arRealAxisAdmin[46].i.Dist:=222.25;
arRealAxisAdmin[46].i.HomeOffset:=HMI_HomeOffsetBelt[6];
arRealAxisAdmin[46].i.Vel:=HMI_BeltVelo[6];
arRealAxisAdmin[46].i.Acc:=HMI_BeltVelo[6]*100;
arRealAxisAdmin[46].i.Dec:=HMI_BeltVelo[6]*100;
//拉膜伺服
arRealAxisAdmin[47].i.Pos:=HMI_PullerPara[1];
arRealAxisAdmin[47].i.Dist:=HMI_PullerPara[1];
arRealAxisAdmin[47].i.JogVel:=HMI_PullerPara[2];
arRealAxisAdmin[47].i.JogAcc:=HMI_PullerPara[3];
arRealAxisAdmin[47].i.JogDec:=HMI_PullerPara[3];
arRealAxisAdmin[47].i.Vel:=HMI_PullerPara[2];
arRealAxisAdmin[47].i.Acc:=HMI_PullerPara[3];
arRealAxisAdmin[47].i.Dec:=HMI_PullerPara[3];
//皮带7 
arRealAxisAdmin[48].i.Dist:=150;
arRealAxisAdmin[48].i.HomeOffset:=HMI_HomeOffsetBelt[7];
arRealAxisAdmin[48].i.Vel:=HMI_BeltVelo[7];
arRealAxisAdmin[48].i.Acc:=HMI_BeltVelo[7]*100;
arRealAxisAdmin[48].i.Dec:=HMI_BeltVelo[7]*100;
//推瓶伺服
END_ACTION

ACTION SR05_Manual:
IF (Ref_MachineStateModel.Sts_Stopped OR Ref_MachineStateModel.Sts_Held) AND NOT  glb_bModeSwitch_UN01 THEN

	FOR i:=1 TO 40 DO
      arDropCylinder[i].i.ActiveIn:=FALSE;
	  arDropCylinder[i].i.ActiveOut:=FALSE;
	END_FOR
	
	FOR i:= 1 TO 20 DO
		arPackCylinder[i].i.ActiveIn:=FALSE;
		arPackCylinder[i].i.ActiveOut:=FALSE;	
    END_FOR
	
	FOR i:= 1 TO 10 DO
		arPackVacuum[i].i.ActiveIn:=FALSE;	
    END_FOR	


    FOR i:= 1 TO 40 DO
		IF HMI_ClearCounter[i] THEN
		   arRealAxisAdmin[i].i.Enable:=TRUE;
		END_IF
	END_FOR

    FOR i:= 1 TO 50 DO
	    arRealAxisAdmin[i].i.Mode:=1;
	END_FOR
ELSE
	 FOR i:=1 TO 32 DO 
		 FOR j:=1 TO 8 DO
			 DO_[i,j].ON:=FALSE;
			 DO_[i,j].Off:=FALSE;					 
		 END_FOR
	 END_FOR
	 FOR i:=50 TO 57 DO 
		 FOR j:=1 TO 8 DO
			 DO_[i,j].on:=FALSE;
			 DO_[i,j].Off:=FALSE;
		 END_FOR
	 END_FOR
	 FOR i:=1 TO 37 DO 
		 FOR j:=1 TO 8 DO
			 Di_[i,j].on:=FALSE;
			 Di_[i,j].Off:=FALSE;
		 END_FOR
	 END_FOR	 
	 
     FOR i:= 1 TO 50 DO
	     arRealAxisAdmin[i].i.Mode:=0;
		 HMI_AxisView[i].MoveReal:=FALSE;
	 END_FOR
	 HMI_AutoCut:=FALSE;
	 HMI_CutCnt:=0;
END_IF

//手动防护位
HMI_ManualInhibit[0]:=NOT arPackCylinder[1].i.InSensor OR NOT arPackCylinder[2].i.InSensor OR NOT arPackCylinder[3].i.InSensor  
OR NOT arPackCylinder[4].i.InSensor OR NOT arPackCylinder[5].i.InSensor OR NOT arPackCylinder[6].i.InSensor 
OR NOT arPackCylinder[7].i.InSensor OR NOT arPackCylinder[12].i.InSensor OR NOT arPackCylinder[15].i.InSensor
OR NOT arPackCylinder[16].i.InSensor OR NOT arPackCylinder[17].i.InSensor 
OR NOT arPackCylinder[10].i.InSensor OR NOT arPackCylinder[11].i.InSensor OR NOT arPackCylinder[41].i.InSensor ;

HMI_ManualInhibit[1]:=  arDropBufferCyclinder[1].i.InSensor AND arDropBufferCyclinder[2].i.InSensor;

CASE iAutoCut OF 
	0: IF HMI_AutoCut AND arRealAxisAdmin[47].o.PowerOn AND arRealAxisAdmin[46].o.PowerOn AND NOT glb_bModeSwitch_UN01 
       AND HMI_CutCnt>0 THEN
		  iAutoCut:=1;
		  iCutCnt:=iCutCnt+1;
	   END_IF
	1: 
       HMI_AxisView[47].MoveReal:=TRUE;
	   iAutoCut:=2;
	2: 
       tonAutoCut(IN:= TRUE, PT:= T#3S, Q=> , ET=> ); 
	   IF tonAutoCut.Q THEN 
	       tonAutoCut(IN:= FALSE, PT:= T#3S, Q=> , ET=> ); 
           iAutoCut:=3;	   
	   END_IF

    3:
	   HMI_AxisView[47].MoveReal:=FALSE;
       DO_[31,6].ON:=TRUE;
	   iAutoCut:=4;	
    4:
       tonAutoCut(IN:= TRUE, PT:= T#2S, Q=> , ET=> ); 
	   IF tonAutoCut.Q THEN 
	       tonAutoCut(IN:= FALSE, PT:= T#2S, Q=> , ET=> ); 
           iAutoCut:=5;	   
	   END_IF	
	   
    5: DO_[31,6].ON:=FALSE;
	   iAutoCut:=6;	
    6: 	  
       tonAutoCut(IN:= TRUE, PT:= T#3S, Q=> , ET=> ); 
	   IF tonAutoCut.Q THEN 
	       tonAutoCut(IN:= FALSE, PT:= T#3S, Q=> , ET=> ); 
           iAutoCut:=7;	   
	   END_IF	
    7: 
 	   IF icutcnt> HMI_cutCnt THEN
		  iAutoCut:=8; 
	   ELSE 
	      iAutoCut:=0; 
	   END_IF
	8:   
       HMI_AxisView[46].MoveReal:=TRUE;
	   iAutoCut:=9;	  
 
	9:
       tonAutoCut(IN:= TRUE, PT:= T#2S, Q=> , ET=> ); 
	   IF tonAutoCut.Q THEN 
	       tonAutoCut(IN:= FALSE, PT:= T#2S, Q=> , ET=> ); 
           iAutoCut:=10;	   
	   END_IF	
	   
	10:
	   icutcnt:=0;
       HMI_AxisView[46].MoveReal:=FALSE;
	   iAutoCut:=0;		   
	   
END_CASE


tonCounterAirOpen(IN:= glb_bCounterAirValve_UN01 , PT:= T#3S, Q=> , ET=> );
IF tonCounterAirOpen.Q THEN
   glb_bPackAirValve_UN01:=TRUE;
END_IF


IF HMI_DisableCntAlarmAll THEN
	FOR  i:=1 TO 40 DO
		HMI_SkipCntAlarm[i]:=TRUE;
	END_FOR
END_IF

IF HMI_EnbaleCntAlarmAll THEN
	FOR  i:=1 TO 40 DO
		HMI_SkipCntAlarm[i]:=FALSE;
	END_FOR	
END_IF

IF HMI_DisableCntAlarmAll2 THEN
	FOR  i:=1 TO 40 DO
		HMI_CntCheck[i]:=TRUE;
	END_FOR
END_IF

IF HMI_EnbaleCntAlarmAll2 THEN
	FOR  i:=1 TO 40 DO
		HMI_CntCheck[i]:=FALSE;
	END_FOR	
END_IF
END_ACTION

ACTION SR90_SafetyReset:
CASE iSafetyResetSeq OF
	0: IF glb_bSafetyReset THEN
		  iSafetyResetSeq:=10;
	   END_IF
	10: 	
		IF glb_arSafeRelayNo_UN01[1] OR tonSafetyReset.Q  THEN
		    iSafetyResetSeq:=20;
		END_IF
	20:	
		FOR i:=1 TO 64 DO
		    arRealAxisAdmin[i].i.Reset:= TRUE ;
			iSafetyResetSeq:=30;
		END_FOR		
	30:
	    IF tonSafetyReset.Q THEN
		   FOR i:=1 TO 64 DO
		       arRealAxisAdmin[i].i.Reset:= FALSE ;	
	       END_FOR	
		   glb_bSafetyreset:=FALSE;
		   iSafetyResetSeq:=0;
		END_IF
	
END_CASE

tonSafetyReset(IN:=glb_bSafetyreset , PT:=T#3S , Q=> , ET=> );

	
IF glb_arSafeRelayNo_UN01[1] THEN
	glb_bAllSafetyOk:=TRUE;
	ELSE 
	glb_bAllSafetyOk:=FALSE;
END_IF
END_ACTION

ACTION SR91_OEE:
HMI_OEEView.Active:=TRUE;
IF HMI_OEEView.Active THEN
   IF rtGoodCount.Q THEN	
      HMI_OEEView.GoodCount:= HMI_OEEView.GoodCount+7;	
   END_IF 
   IF rtNoGoodCount.Q THEN
	  HMI_OEEView.NoGoodCount:= HMI_OEEView.NoGoodCount+7;
   END_IF
  
END_IF

rtGoodCount(CLK:= glb_digoodFlag_UN01.11, Q=> );
rtNoGoodCount(CLK:= glb_diNogoodFlag_UN01.11 , Q=> );

IF HMI_OEEView.Reset THEN
   HMI_OEEView.GoodCount:=0;
   HMI_OEEView.NoGoodCount:=0;	
END_IF


HMI_OEEView.DesignSpeed:= 7.5;
HMI_OEEView.Performance:=HMI_OEEView.AverageSpeed/HMI_OEEView.DesignSpeed*100;


aoiActiveTotalTime(
	bEnable:= HMI_OEEView.Active, 
	bReset:= HMI_OEEView.Reset, 
	diSecond=> , 
	diMinute=> , 
	diHour=> , 
	diTotalSecond=> , 
	diTotalMinute=> HMI_OEEView.PlannedTime, 
	diTotalHour=> );

aoiWorkTotalTime(
	bEnable:= HMI_OEEView.Active AND Ref_MachineStateModel.Sts_Execute, 
	bReset:= HMI_OEEView.Reset, 
	diSecond=> , 
	diMinute=> , 
	diHour=> , 
	diTotalSecond=> , 
	diTotalMinute=> HMI_OEEView.UsableTime, 
	diTotalHour=> );

aoi10MinuteTime(
	bEnable:= bEn10Minute OR TRUE, 
	bReset:= bReset10Minute, 
	diSecond=> , 
	diMinute=> , 
	diHour=> , 
	diTotalSecond=> , 
	diTotalMinute=> , 
	diTotalHour=> );
	

HMI_OEEView.AverageSpeed:=DINT_TO_REAL(glb_TransferCnt)*7/DINT_TO_REAL(aoiWorkTotalTime.diTotalMinute);

	
IF	aoiActiveTotalTime.diTotalMinute>0 THEN
    HMI_OEEView.Usability:= DINT_TO_REAL(aoiWorkTotalTime.diTotalMinute)/DINT_TO_REAL(aoiActiveTotalTime.diTotalMinute)*100;
ELSE
    HMI_OEEView.Usability:= 0;
END_IF	

IF (HMI_OEEView.NoGoodCount+HMI_OEEView.GoodCount)> 0 THEN
    HMI_OEEView.Quality:=DINT_TO_REAL(HMI_OEEView.GoodCount)/(DINT_TO_REAL(HMI_OEEView.NoGoodCount)+DINT_TO_REAL(HMI_OEEView.GoodCount))*100;
ELSE
	HMI_OEEView.Quality:=0;
END_IF

HMI_OEEView.OEE:=(HMI_OEEView.Quality/100*HMI_OEEView.Usability/100*HMI_OEEView.Performance/100)*100;
END_ACTION

ACTION SR99_FaultClear:
CASE iFaultClearSeq OF
	0: 
		IF bClearAllFault THEN
		   iFaultClearSeq:=10;
		END_IF
	   
	10: 	
	//    IF NOT glb_bAirFeedback_UN01[2] THEN
	//		glb_bCounterAirValve_UN01:=FALSE;
	//	END_IF
	
	//	IF NOT glb_bAirFeedback_UN01[1] THEN
	//		glb_bPackAirValve_UN01:=FALSE;
	//	END_IF
		
		glb_MembraneAlarm:=FALSE;
		FOR i:=1 TO 50 DO
			IF arRealAxisAdmin[i].o.Error  THEN
			   arRealAxisAdmin[i].i.Reset:= TRUE ;
			END_IF
			IF arVirtualAxisAdmin[i].o.Error THEN
			   arVirtualAxisAdmin[i].i.Reset:= TRUE ;
			END_IF
		END_FOR
	
		FOR j:=1 TO 40 DO
			IF arDropCylinder[j].o.Error THEN
		       arDropCylinder[j].i.Reset:=TRUE;
			END_IF
			IF arCounters[j].Error THEN
			   arCounters[j].Clear:=TRUE;
			END_IF
		END_FOR
	    FOR j:=1 TO 50 DO
 			IF arPackCylinder[j].o.Error THEN
		       arPackCylinder[j].i.Reset:=TRUE;
			END_IF
			IF arPackVacuum[j].o.Error THEN
		       arPackVacuum[j].i.Reset:=TRUE;
			END_IF  
		END_FOR		
		
		FOR j:=1 TO 8 DO
			arHeat_AOI[j].Reset:=TRUE;
		END_FOR
        arDropBufferCyclinder[1].i.Reset:=TRUE;
		arDropBufferCyclinder[2].i.Reset:=TRUE;
	    iFaultClearSeq:=20;

	20:
		HMI_StopEvent[5].ID[20]:=FALSE;
		HMI_StopEvent[5].ID[21]:=FALSE;
		HMI_StopEvent[5].ID[22]:=FALSE;
		HMI_StopEvent[5].ID[23]:=FALSE;
		HMI_StopEvent[5].ID[24]:=FALSE;
		HMI_StopEvent[5].ID[25]:=FALSE;
		HMI_StopEvent[5].ID[26]:=FALSE;
	
	   IF  tonFaultClear.Q THEN 
			FOR i:=1 TO 50 DO
				 arRealAxisAdmin[i].i.Reset:= FALSE ;
				 arVirtualAxisAdmin[i].i.Reset:= FALSE ;
			END_FOR
			FOR j:=1 TO 40 DO
				arDropCylinder[j].i.Reset:=FALSE;
			    arCounters[j].Clear:=FALSE;				
			END_FOR
			FOR j:=1 TO 50 DO
				arPackCylinder[j].i.Reset:=FALSE;
				arPackVacuum[j].i.Reset:=FALSE;
			END_FOR			
			
			FOR j:=1 TO 8 DO
				arHeat_AOI[j].Reset:=FALSE;
			END_FOR
		    HMI_PrinterFault:=FALSE;
			
		    HMI_StopEvent[0].ID[6]:=FALSE;
		    HMI_StopEvent[0].ID[7]:=FALSE;
			
		//	glb_bPackAirValve_UN01:=TRUE;
		//	glb_bCounterAirValve_UN01:=TRUE;
		
		    arDropBufferCyclinder[1].i.Reset:=FALSE;
		    arDropBufferCyclinder[2].i.Reset:=FALSE;
		
			HMI_AlarmMute:=FALSE;
			bClearAllFault:=FALSE;
			iFaultClearSeq:=0;
       END_IF
	   
END_CASE

tonFaultClear(IN:=bClearAllFault , PT:=T#500MS , Q=> , ET=> );
END_ACTION

ACTION UP01_PackML:
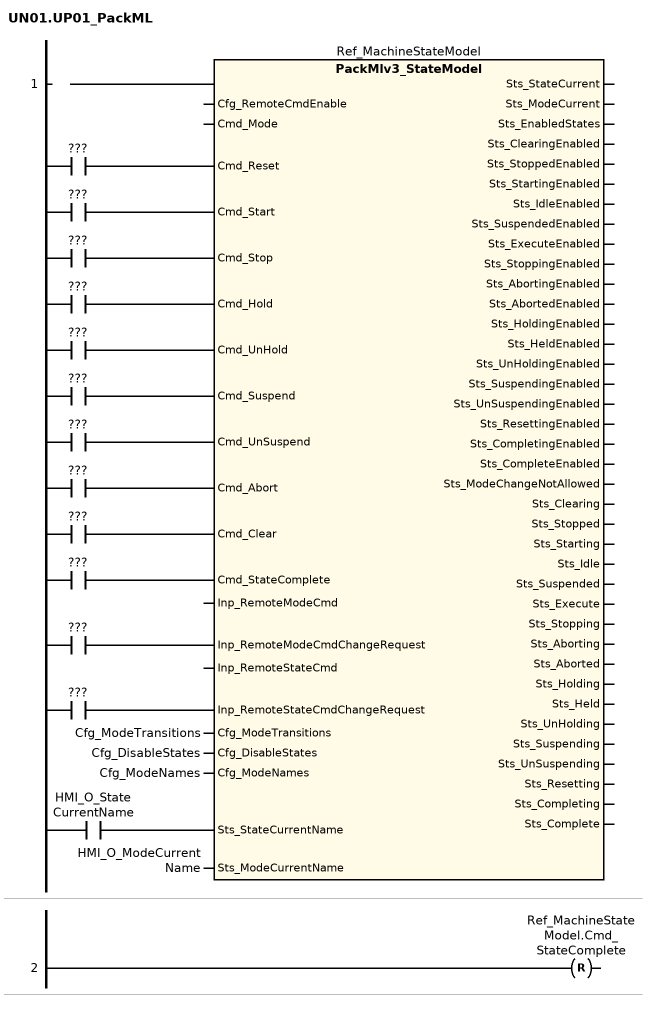
// NETWORK 1
Ref_MachineStateModel(
    Cfg_ModeTransitions := Cfg_ModeTransitions,
    Cfg_DisableStates := Cfg_DisableStates,
    Cfg_ModeNames := Cfg_ModeNames,
    Sts_StateCurrentName := HMI_O_StateCurrentName,
    Sts_ModeCurrentName := HMI_O_ModeCurrentName); // PackMlv3_StateModel

// NETWORK 2
Ref_MachineStateModel.Cmd_StateComplete R= TRUE;
END_ACTION

ACTION UP02_StateComplete:
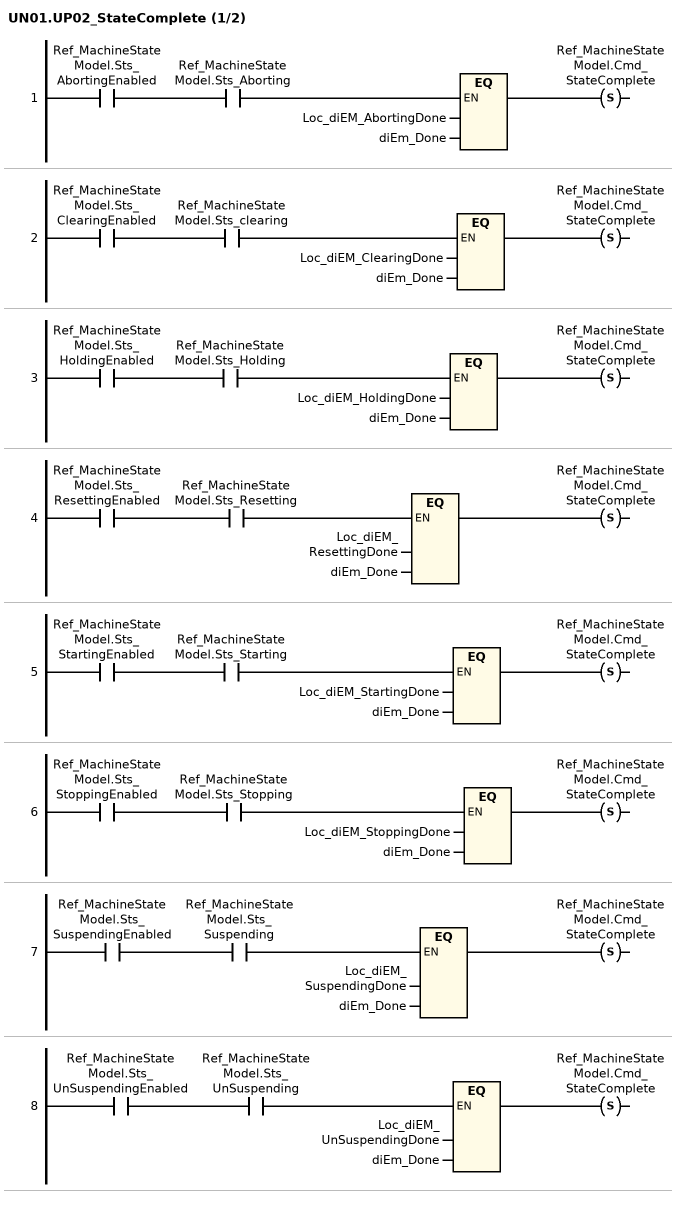
// NETWORK 1
Ref_MachineStateModel.Cmd_StateComplete S= Ref_MachineStateModel.Sts_AbortingEnabled AND Ref_MachineStateModel.Sts_Aborting AND Loc_diEM_AbortingDone = diEm_Done;

// NETWORK 2
Ref_MachineStateModel.Cmd_StateComplete S= Ref_MachineStateModel.Sts_ClearingEnabled AND Ref_MachineStateModel.Sts_clearing AND Loc_diEM_ClearingDone = diEm_Done;

// NETWORK 3
Ref_MachineStateModel.Cmd_StateComplete S= Ref_MachineStateModel.Sts_HoldingEnabled AND Ref_MachineStateModel.Sts_Holding AND Loc_diEM_HoldingDone = diEm_Done;

// NETWORK 4
Ref_MachineStateModel.Cmd_StateComplete S= Ref_MachineStateModel.Sts_ResettingEnabled AND Ref_MachineStateModel.Sts_Resetting AND Loc_diEM_ResettingDone = diEm_Done;

// NETWORK 5
Ref_MachineStateModel.Cmd_StateComplete S= Ref_MachineStateModel.Sts_StartingEnabled AND Ref_MachineStateModel.Sts_Starting AND Loc_diEM_StartingDone = diEm_Done;

// NETWORK 6
Ref_MachineStateModel.Cmd_StateComplete S= Ref_MachineStateModel.Sts_StoppingEnabled AND Ref_MachineStateModel.Sts_Stopping AND Loc_diEM_StoppingDone = diEm_Done;

// NETWORK 7
Ref_MachineStateModel.Cmd_StateComplete S= Ref_MachineStateModel.Sts_SuspendingEnabled AND Ref_MachineStateModel.Sts_Suspending AND Loc_diEM_SuspendingDone = diEm_Done;

// NETWORK 8
Ref_MachineStateModel.Cmd_StateComplete S= Ref_MachineStateModel.Sts_UnSuspendingEnabled AND Ref_MachineStateModel.Sts_UnSuspending AND Loc_diEM_UnSuspendingDone = diEm_Done;

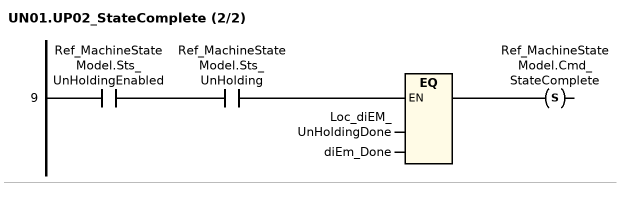
// NETWORK 9
Ref_MachineStateModel.Cmd_StateComplete S= Ref_MachineStateModel.Sts_UnHoldingEnabled AND Ref_MachineStateModel.Sts_UnHolding AND Loc_diEM_UnHoldingDone = diEm_Done;
END_ACTION

END_PROGRAM

(* stored: Version 1.1.0.1, ProductVersion 3.1.4024.6
   POU UN01: Id {a96c2e98-15ed-4710-a682-9999665d2585}, SpecialFunc None
   Action CM01_OperationLocal: Id {dff45118-d795-4716-bdc6-ad799f5e59b7}
   Action CM02_ConditionsModules: Id {da4a938a-8219-4f45-b1ac-86701ae4763d}
   Action CM03_Cylinder: Id {6d7500e9-d9b1-4a89-86b1-8a4920e98324}
   Action CM04_Vacuum: Id {5e4ae751-7643-4662-a961-8c1abf670331}
   Action CM05_Sensor: Id {c9ea1b24-9952-474f-9bc9-b6b369adf20f}
   Action CM06_Heat: Id {42b1757a-8a29-4c78-b1d7-18b856d0f0ac}
   Action CM07_Counters: Id {c6109522-4e52-4e09-9fa0-3a70d3590e76}
   Action CM10_LightStatus: Id {f1a2fc42-0a34-4ceb-8734-10a495a9dcf3}
   Action SR01_Initialize: Id {e3f8d4f1-7249-43dd-82f4-f3aa9b73d1cf}
   Action SR02_Recipe: Id {97908948-cd99-4066-b1a3-b4f07a0cffee}
   Action SR03_FaultHandler: Id {b7f7c2b4-b35e-4964-97ca-7884fde86859}
   Action SR04_Parameter: Id {3ef137e3-6494-42e9-b13a-3a5700d6a5aa}
   Action SR05_Manual: Id {52b80dfd-0e99-4c9c-83b7-0efba1b21f76}
   Action SR90_SafetyReset: Id {2f37013d-0e28-4cd7-8e9b-3854564c9c8b}
   Action SR91_OEE: Id {57267c99-8089-4fbf-83e0-4621734d5fdd}
   Action SR99_FaultClear: Id {6d43a824-e65a-4707-aa24-ba03da90ea45}
   Action UP01_PackML: Id {17ac2d4b-f212-458b-af30-289d64f20804}
   Action UP02_StateComplete: Id {9611c9b0-5cf6-4bdc-93f3-c1f1606ad42e} *)
